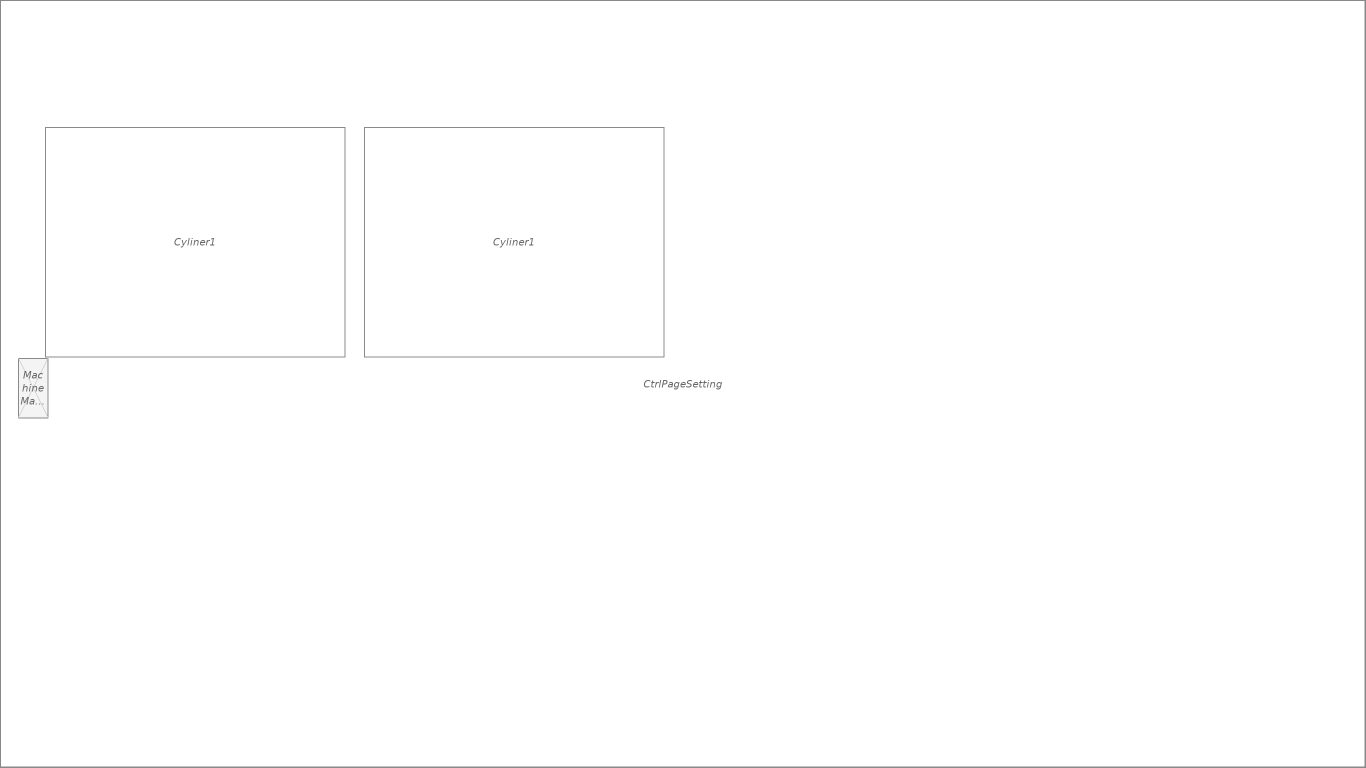
VISUALIZATION PageSetting_AcquireLoad_2  // 1366x768
    Frame (0,0 1366x768)
        shows CtrlPageSetting()
    Frame (45,127 300x230)
        shows Cyliner1(System := G_stSystem, Cylinder := G_arrCylinder[E_Cylinder.AcquirePrevent2], CylinderData := G_arrCylinderData[E_Cylinder.AcquirePrevent2])
    Image (18,358 30x60), image: MachineManage.ImagePool.prev
        OnMouseClick: change screen: PageSetting_AcquireLoad
    Frame (364,127 300x230)
        shows Cyliner1(System := G_stSystem, Cylinder := G_arrCylinder[E_Cylinder.AcquirePrevent0], CylinderData := G_arrCylinderData[E_Cylinder.AcquirePrevent0])
END_VISUALIZATION

(* stored: Version 1.1.0.1, ProductVersion 3.1.4024.3
   Visu PageSetting_AcquireLoad_2: Id {dd3f6614-219b-4f43-b0c5-412436f11c13} *)
